(* IEC 61131-3 sources: pandora/pandora/aws-platform-main/aws-platform-main/src/Utils/Timer, 2 files *)

(* ---- ITimer.st ---- *)
NAMESPACE Esab.Utils.Timer

    INTERFACE ITimer
        /// Cyclic execute
        METHOD Execute
            VAR_INPUT
                signal : BOOL;
                duration : LTIME;
            END_VAR
        END_METHOD

        /// Returns TRUE if this timer is expired
        METHOD Expired : BOOL
        END_METHOD

        /// Returns the elapsed time
        METHOD ElapsedTime : LTIME
        END_METHOD
    END_INTERFACE

END_NAMESPACE

(* ---- OnDelay.st ---- *)
NAMESPACE Esab.Utils.Timer

    CLASS OnDelay IMPLEMENTS ITimer
        VAR PRIVATE
            _onDelay : System.Timer.OnDelay;
        END_VAR

        METHOD PUBLIC Execute
            VAR_INPUT
                signal : BOOL;
                duration : LTIME;
            END_VAR

            _onDelay(signal, duration);
        END_METHOD

        METHOD PUBLIC Expired : BOOL
            Expired := _onDelay.output;
        END_METHOD

        METHOD PUBLIC ElapsedTime : LTIME
            ElapsedTime := _onDelay.elapsedTime;
        END_METHOD
    END_CLASS

END_NAMESPACE
